{attribute 'GeneratedUsingTerminal: EP4374-0002-0016'}
{attribute addProperty BoxType "EP4374-0002-0016"}
{attribute addProperty Id "AI_TxPDO_Map_Standard_Channel_1AT %I*AI_TxPDO_Map_Standard_Channel_A8DF64E310AI_TxPDO_Map_Standard_Channel_2AT %I*AI_TxPDO_Map_Standard_Channel_A8DF64E310AO_RxPDO_Map_Channel_3AT %Q*AO_RxPDO_Map_Channel_BA7EBB7C2AO_RxPDO_Map_Channel_4AT %Q*AO_RxPDO_Map_Channel_BA7EBB7C2WcStateAT %I*WcState_9091E0EB2InfoDataAT %I*InfoData_32EB74EA10"}
{attribute addProperty CRC "1289502765"}
{attribute addProperty Size "36"}
TYPE EP4374_4CDC402D :
STRUCT
	{attribute addProperty Name "AI_TxPDO_Map_Standard_Channel_1"}
	AI_TxPDO_Map_Standard_Channel_1 : AI_TxPDO_Map_Standard_Channel_A8DF64E3;
	{attribute addProperty Name "AI_TxPDO_Map_Standard_Channel_2"}
	AI_TxPDO_Map_Standard_Channel_2 : AI_TxPDO_Map_Standard_Channel_A8DF64E3;
	{attribute addProperty Name "AO_RxPDO_Map_Channel_3"}
	AO_RxPDO_Map_Channel_3 : AO_RxPDO_Map_Channel_BA7EBB7C;
	{attribute addProperty Name "AO_RxPDO_Map_Channel_4"}
	AO_RxPDO_Map_Channel_4 : AO_RxPDO_Map_Channel_BA7EBB7C;
	{attribute addProperty Name "WcState"}
	WcState : WcState_9091E0EB;
	{attribute addProperty Name "InfoData"}
	InfoData : InfoData_32EB74EA;
END_STRUCT
END_TYPE

(* stored: Version 1.2.0.0, ProductVersion 3.1.4024.9
   DUT EP4374_4CDC402D: Id {4369a568-7726-4dcc-bfde-fab8c7d842f2} *)
